FUNCTION_BLOCK Button (* Composite Function Block Type *)
  (* Standard: 61499-2 *)
  (* Version 0.0, 5/25/2016, Andrei, nxtControl GmbH, template *)
  PACKAGE Main;
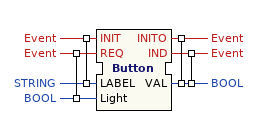
  EVENT_INPUT
    INIT WITH LABEL; (* Initialization Request *)
    REQ WITH Light;
  END_EVENT
  EVENT_OUTPUT
    INITO WITH VAL; (* Initialization Confirm *)
    IND WITH VAL; (* Execution Confirmation *)
  END_EVENT
  VAR_INPUT
    LABEL : STRING;
    Light : BOOL;
  END_VAR
  VAR_OUTPUT
    VAL : BOOL;
  END_VAR
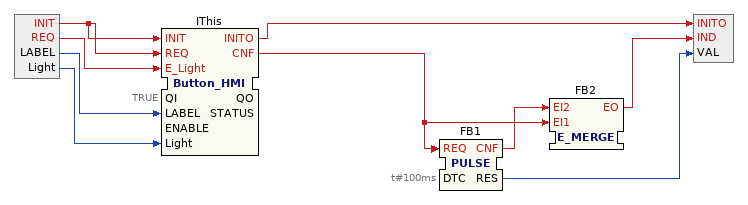
  FBS
    FB1 : PULSE(DTC := t#100ms);
    IThis : Button_HMI(QI := TRUE);
    FB2 : E_MERGE;
  END_FBS
  EVENT_CONNECTIONS
    FB1.CNF TO FB2.EI2;
    FB2.EO TO IND;
    INIT TO IThis.INIT;
    INIT TO IThis.REQ;
    REQ TO IThis.E_Light;
    IThis.INITO TO INITO;
    IThis.CNF TO FB2.EI1;
    IThis.CNF TO FB1.REQ;
  END_CONNECTIONS
  DATA_CONNECTIONS
    FB1.RES TO VAL;
    LABEL TO IThis.LABEL;
    Light TO IThis.Light;
  END_CONNECTIONS
END_FUNCTION_BLOCK
